(* PLC project add_syrup, Dassault Systèmes ControlBuild 2024x Refresh1 *)
(* stored: creationDateTime 2024-04-12T14:05:56-01:00 *)

FUNCTION_BLOCK copie_batch.add_syrup
  VAR_INPUT
    flowSyrup1 : REAL := 0.0;
    flowSyrup2 : REAL := 0.0;
    flowSyrup3 : REAL := 0.0;
  END_VAR
  VAR_OUTPUT
    flow : REAL := 0.0;
  END_VAR

IF (flowSyrup1+flowSyrup2+flowSyrup3>0.0) THEN
	flow := flowSyrup1+flowSyrup2+flowSyrup3;
ELSE
	flow := 0.0;
END_IF;
END_FUNCTION_BLOCK
